// TIA Portal V18 export
TYPE "UDT_HWModulesMap"
// stored: IsFailsafeCompliant false
   STRUCT
      cRack : Byte;
      cModule : Byte;
      wLaddr1 : Word;
      wLaddr2 : Word;
      iDiagBuffer : USInt;
      iOwnState : UInt;
      wMaintenanceState : DWord;
      wComponentStateDetail : DWord;
      iOperatingState : UInt;
   END_STRUCT;
END_TYPE
